/// This the main class of the library. It represents a OpenWeatherMap app and
/// is tied to a unique API token. When constructing the object it is mandatory to pass
/// an `app-token``.
///
/// Here's a simple example, which requests the current data for 'Innsbruck, AT'.
/// The actual action of sending the notification is triggered by [RequestWeatherByZipCodeAsync](xref:OpenWeatherMap.OpenWeatherMapClient#RequestWeatherByZipCodeAsync).
/// The ´Async´ Suffix in this method indicates that this action has to be waited for by checking for ´NOT _openWeatherMapClient.Busy´ before
/// sending another request.
///
/// ```sti
/// PROGRAM MAIN
/// VAR
///   _send : BOOL; // boolean, which can be triggered to send a message
///   _openWeatherMapClient : OpenWeatherMap.OpenWeatherMapClient('<your_openweathermap_apptoken>'); 
/// END_VAR
/// ```
/// ```std
/// IF _send
/// THEN
///   _send := FALSE;
///   _openWeatherMapClient.RequestWeatherByZipCodeAsync('6020', 'AT');
/// END_IF
///
/// _openWeatherMapClient.Cyclic();
/// ```
{attribute 'conditionalshow_all_locals'}
{attribute 'no_explicit_call' := 'This FB is a CLASS and must be accessed using methods and/or properties'}
{attribute 'hide_all_locals'}
FUNCTION_BLOCK OpenWeatherMapClient
VAR
  _busy : BOOL;
  _error : BOOL;
  _errorMessage : STRING(255);
  
  _request : OpenWeatherMapRequest;
  _response : OpenWeatherMapResponse;
  
  _server : Tc2_System.ADSRDWRTEX;
END_VAR
VAR CONSTANT
  _defaultHost : STRING := '127.0.0.1.1.1';
  _defaultPort : UINT := 25734;
END_VAR

/// This property can be used to check if the client is ready for sending request. If the client is not 
/// ready or an error occurs during sending (e.g. not internet connection, OpenWeatherMap Twincat Service is not running, ...)
/// the property [Error](xref:OpenWeatherMap.OpenWeatherMapClient#Error) returns `true`.
{attribute 'monitoring' := 'call'}
PROPERTY Busy : BOOL
GET
Busy := _busy;
END_GET
SET // PROTECTED
_busy := Busy;

IF _busy
THEN
  _error := FALSE;
END_IF
END_SET
END_PROPERTY

/// This method has to be called cyclically and takes care of the communication with the `OpenWeatherMap Twincat Service`, which is reached 
/// via [Host](xref:OpenWeatherMap.OpenWeatherMapClient#Host) and [Port](xref:OpenWeatherMap.OpenWeatherMapClient#Port).
/// You can use the properties [Busy](xref:OpenWeatherMap.OpenWeatherMapClient#Busy) and [Error](xref:OpenWeatherMap.OpenWeatherMapClient#Error) to check weather an
/// operation was successful (`NOT Busy AND NOT Error`) or failed (`Error`), respectively.
METHOD Cyclic
VAR_INST
  errorTrig : Tc2_Standard.R_TRIG;
END_VAR
IF NOT Busy
THEN
  RETURN;
END_IF

_server(IDXOFFS:=0, 
        WRITELEN:=SIZEOF(_request),
        SRCADDR:=ADR(_request),
        WRTRD:=TRUE, 
        TMOUT:=T#5S,
        ERR=>,
        BUSY=>,
        ERRID=>);
  
IF _server.ERR // fallback to proxy
THEN
  Error := TRUE;
  ErrorMessage := Tc2_Standard.CONCAT('Error Code: ', UDINT_TO_STRING(_server.ERRID));
ELSIF NOT _server.BUSY 
THEN
  Busy := FALSE;

  IF _response.Status = 0
  THEN
    Error := TRUE;
    ErrorMessage := 'No data received';  
  ELSIF _response.Status > 0
  THEN
    Error := TRUE;
    ErrorMessage := _response.Exception;
	END_IF

END_IF
END_METHOD

/// Returns `true` if any error occured when calling an `XXX_Async` method of this object. The details of the error
/// are available by checking the proeprty
{attribute 'monitoring' := 'call'}
PROPERTY Error : BOOL
GET
Error := _error;
END_GET
SET // PROTECTED
_error := Error;

IF _error
THEN
  _busy := FALSE;
END_IF
END_SET
END_PROPERTY

/// Only valid if `Error=TRUE`, returns the explanation why the call of an `XXX_Async` method failed.
{attribute 'monitoring' := 'call'}
PROPERTY ErrorMessage : STRING(255)
GET
IF _error
THEN
  ErrorMessage := _errorMessage;
END_IF
END_GET
SET // PROTECTED
_errorMessage := ErrorMessage;
END_SET
END_PROPERTY

METHOD FB_init : BOOL
VAR_INPUT
	bInitRetains : BOOL; // if TRUE, the retain variables are initialized (warm start / cold start)
	bInCopyCode : BOOL;  // if TRUE, the instance afterwards gets moved into the copy code (online change)
  
  /// The OpenWeatherMap API token
  token : STRING;
END_VAR
THIS^.Token := token;
THIS^.Host := _defaultHost;
THIS^.Port := _defaultPort;

Reset();
END_METHOD

/// Returns the AMS Net Id of the `OpenWeatherMap Twincat Service`. Defaults to localhost
PROPERTY Host : STRING
GET
Host := _server.NETID;
END_GET
SET
_server(WRTRD := FALSE,
       NETID := Host,
       BUSY=>,
       ERR=>,
       ERRID=>);
END_SET
END_PROPERTY

PROPERTY Port : UINT
GET
Port := _server.PORT;
END_GET
SET
_server(WRTRD := FALSE,
       PORT := Port,
       BUSY=>,
       ERR=>,
       ERRID=>);
END_SET
END_PROPERTY

METHOD RequestWeatherByZipCodeAsync
VAR_IN_OUT CONSTANT
  zipCode : STRING(9);
  countryCode : STRING(4);
END_VAR
IF NOT Busy
THEN
  _request.ZipCodeLength := Tc2_Standard.LEN(zipCode);
  _request.ZipCode := zipCode;
  _request.CountryCodeLength := Tc2_Standard.LEN(countryCode);
  _request.CountryCode := countryCode;
  
  _response.Status := 0;
  
  _server(WRTRD := FALSE,
         IDXGRP:=0,
         DESTADDR:=ADR(_response),
         READLEN:=SIZEOF(_response),
         TMOUT:=TIME#10S,
         BUSY=>,
         ERR=>,
         ERRID=>);    
  Busy := TRUE;
ELSE
  Error := TRUE;
  _errorMessage := 'Client can not executed parallel requests!';
END_IF
END_METHOD

/// Resets client to default values
METHOD Reset
VAR
  token : STRING;
  host : STRING;
  port : UINT;  
END_VAR
token := THIS^.Token;
host := THIS^.Host;
port := THIS^.Port;

Tc2_System.MEMSET(ADR(_request), 0, SIZEOF(_request));

THIS^.Token := token;
THIS^.Host := _defaultHost;
THIS^.Port := _defaultPort;
END_METHOD

PROPERTY Token : STRING
GET
Token := _request.Token;
END_GET
SET
_request.Token := Token;
_request.TokenLength := Tc2_Standard.LEN(_request.Token);
END_SET
END_PROPERTY

{attribute 'monitoring' := 'call'}
PROPERTY Weather : REFERENCE TO OpenWeatherMapResponse
GET
IF _busy OR_ELSE _response.Status = 0
THEN
  Weather REF= 0;
  RETURN;
END_IF

Weather REF= _response;
END_GET
END_PROPERTY

END_FUNCTION_BLOCK

(* stored: Version 1.1.0.1, ProductVersion 3.1.4024.12
   POU OpenWeatherMapClient: Id {7e1e9724-26e2-0084-1004-42ca9b5de5a8}, SpecialFunc None
   Property Busy: Id {72c62e30-e885-4eb2-98b1-f1d26e618bab}
   Get Get: Id {638df4c4-ce17-46ec-9ad7-929d45026307}
   Set Set: Id {72c23c85-7457-4c77-954b-13dc2bbf6698}
   Method Cyclic: Id {426e1ace-8aa7-0373-078f-f6c08bda3162}
   Property Error: Id {e66821e4-2ee0-4372-9ea9-1eb4dd33a529}
   Get Get: Id {e7a38956-1dfd-4ffd-92e4-bca9edabac1a}
   Set Set: Id {32d3bb0b-6ab6-467b-877b-dec253655bc9}
   Property ErrorMessage: Id {fb1419dd-8959-4c52-a678-e27eff869570}
   Get Get: Id {8cc0de4e-82b4-4158-84b4-5f694a2b39d8}
   Set Set: Id {c440d5c4-cbac-45f0-a41e-5d3d4e4bd3d8}
   Method FB_init: Id {35c9eeb9-61ee-4ff2-8c41-88a6a762ab87}
   Property Host: Id {d06b2e65-bd92-4aa0-a8cf-123040bf4d63}
   Get Get: Id {a03127e3-650c-4e7b-943a-977d03c8073e}
   Set Set: Id {c8ced228-6a9e-4ba5-b049-2d5511e74bd0}
   Property Port: Id {6d99f1c3-57ba-40cf-a01f-00d80a87bd49}
   Get Get: Id {62cd6a40-8a44-4f9c-bdf5-2065126bdfe3}
   Set Set: Id {e9a96dd4-dec0-4ef1-bb24-acc78eea7c5b}
   Method RequestWeatherByZipCodeAsync: Id {2514d27a-339b-498f-a48f-770ba2a832fe}
   Method Reset: Id {0f0aec67-27b6-49f3-bec9-7f030e47c04d}
   Property Token: Id {bf5e10e9-5772-4f05-993b-dd3d2d60441b}
   Get Get: Id {d6e8aca1-e3e6-4f04-8a9f-bce9c98cf5a4}
   Set Set: Id {1a083cd8-6ea7-4bd2-9213-fc1474c0c5d4}
   Property Weather: Id {0269ec4f-7f31-45e8-8e2c-80775300eb05}
   Get Get: Id {56d9b21d-c708-4b95-bf8a-68056613ad6d} *)
